{attribute 'qualified_only'}
VAR_GLOBAL
	pCompType		: ARRAY[0..Param.COMP_CAP] OF POINTER TO CompType;
	nCompTypeNo		: UDINT;
	
	pEntity			: POINTER TO BYTE;
	nEntityNo		: UDINT;
END_VAR

(* stored: Version 1.1.0.1
   GVL _ECS: Id {d4183083-62ce-4b2b-bf20-40b7c5bdaf51} *)
